(* IEC 61131-3 sources: CodesysTest/export/SX_1195.dev/Plc Logic/Application/PRJ Specific/Motion/Motors/Applied Motion/Applied Motion TSM34IP-3DG/FB_BaseAppliedMotionMotorEIP.pou/ScaledProfileVelocity.prop, 1 file *)

(* ---- Get.pm.st ---- *)
(*#-#-#-#-#-#-#-#-#-#---Declaration---#-#-#-#-#-#-#-#-#-#-#-#-#*)

VAR
END_VAR
VAR CONSTANT
	UNITS_PER_ROTATION : REAL := 4.0;
	RPS_TO_RPM : REAL := 60;
END_VAR(*#-#-#-#-#-#-#-#-#-#---Implementation---#-#-#-#-#-#-#-#-#-#-#-#-#*)

ScaledProfileVelocity := FPU.CeilF(profileVelocity * rotationsPerInch * UNITS_PER_ROTATION * RPS_TO_RPM);
